FUNCTION_BLOCK StackControl1
  (* Standard: 61499-2 *)
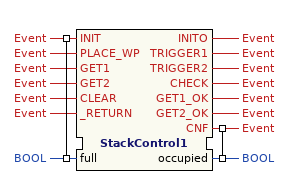
  EVENT_INPUT
    INIT WITH full;
    PLACE_WP;
    GET1;
    GET2;
    CLEAR;
    _RETURN;
  END_EVENT
  EVENT_OUTPUT
    INITO;
    TRIGGER1;
    TRIGGER2;
    CHECK;
    GET1_OK;
    GET2_OK;
    CNF WITH occupied;
  END_EVENT
  VAR_INPUT
    full : BOOL;
  END_VAR
  VAR_OUTPUT
    occupied : BOOL;
  END_VAR
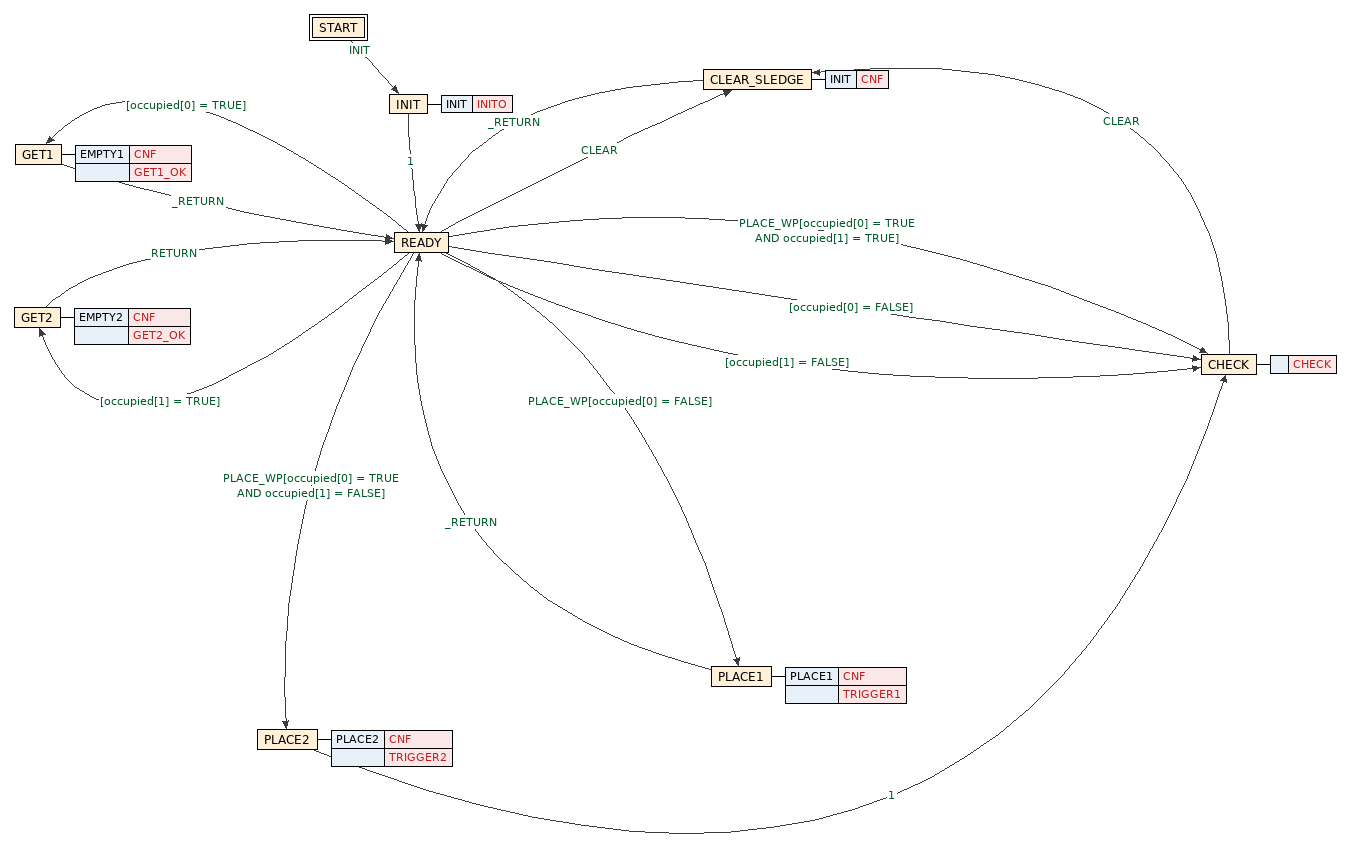
  EC_STATES
    START;
    INIT : INIT -> INITO;
    PLACE1 : PLACE1 -> CNF, -> TRIGGER1;
    CHECK : -> CHECK;
    PLACE2 : PLACE2 -> CNF, -> TRIGGER2;
    GET1 : EMPTY1 -> CNF, -> GET1_OK;
    GET2 : EMPTY2 -> CNF, -> GET2_OK;
    READY;
    CLEAR_SLEDGE : INIT -> CNF;
  END_STATES
  EC_TRANSITIONS
    START TO INIT := INIT;
    INIT TO READY := 1;
    READY TO PLACE1 := PLACE_WP[occupied[0] = FALSE];
    PLACE1 TO READY := _RETURN;
    READY TO CHECK := PLACE_WP[occupied[0] = TRUE AND occupied[1] = TRUE];
    READY TO CLEAR_SLEDGE := CLEAR;
    READY TO CHECK := [occupied[0] = FALSE];
    READY TO CHECK := [occupied[1] = FALSE];
    READY TO PLACE2 := PLACE_WP[occupied[0] = TRUE AND occupied[1] = FALSE];
    PLACE2 TO CHECK := 1;
    READY TO GET1 := [occupied[0] = TRUE];
    GET1 TO READY := _RETURN;
    READY TO GET2 := [occupied[1] = TRUE];
    GET2 TO READY := _RETURN;
    CLEAR_SLEDGE TO READY := _RETURN;
    CHECK TO CLEAR_SLEDGE := CLEAR;
  END_TRANSITIONS
  ALGORITHM INIT IN ST:
IF full THEN&#10;  occupied[0] := TRUE;&#10;  occupied[1] := TRUE;&#10;ELSE&#10;  occupied[0] := FALSE;&#10;  occupied[1] := FALSE;&#10;END_IF;&#10;
  END_ALGORITHM
  ALGORITHM PLACE1 IN ST:
occupied[0] := TRUE;&#10;
  END_ALGORITHM
  ALGORITHM PLACE2 IN ST:
occupied[1] := TRUE;&#10;
  END_ALGORITHM
  ALGORITHM EMPTY1 IN ST:
occupied[0] := FALSE;&#10;
  END_ALGORITHM
  ALGORITHM EMPTY2 IN ST:
occupied[1] := FALSE;&#10;
  END_ALGORITHM
  ALGORITHM READY IN ST:

  END_ALGORITHM
END_FUNCTION_BLOCK
